{attribute 'qualified_only'}
{attribute 'strict'}
// Alarm level enumeration
TYPE E_AlarmLevel :
(
	NONE,
	INFO,
	WARNING,
	ERROR
);
END_TYPE

(* stored: Version 1.1.0.1
   DUT E_AlarmLevel: Id {38e28fc7-5c6d-0ccd-0993-b43dee03152c} *)
